PROGRAM OP160_Initialization_Seq
VAR
	op160_master_reset :BOOL;
	op160_robot_homed  :BOOL;
	op160_ROboProgResetDly   :ton;
END_VAR

IF CR160_MoverREM_Cyl.Position1 AND OP160_SO_Rbt_In_Home AND op160_robot_homed THEN
   OP160_Temp_Home_OK:=TRUE;
ELSE
	OP160_Temp_Home_OK:=FALSE;
END_IF

IF OP160_ErrorActive THEN 
	op160_robot_homed    :=FALSE;
END_IF

CASE OP160_Homing_Seq OF
	
	0: IF (OP160_Auto AND NOT OP160_HomeRunning AND  NOT OP160_ErrorActive AND  NOT 
			OP160_AutoRunning AND NOT OP160_StepRunning	 AND NOT OP160_Temp_Home_OK) THEN
		    OP160_HomeRunning:=TRUE;
		    OP160_Homing_Seq:=10;	
	   END_IF
	   
	10:IF (OP160_HomeRunning AND OP160_HMI_Homing)THEN
		OP160_Homing_Seq:=12;		
		END_IF 
        
	
   12:  OP160_Robo_ProgramReset:=TRUE;
   
		IF NOT OP160_SO_Program_Execute	AND op160_ROboProgResetDly.Q THEN
		OP160_Robo_ProgramReset:=FALSE;			
		OP160_Homing_Seq:=14;	
		END_IF
	
		
	
	14: IF OP160_HomeRunning AND NOT op160_master_reset THEN
		   OP160_Robo_Out6001   :=1;
	       OP160_SI_Homing_Start:=TRUE;
	       OP160_Homing_Seq:=15;
	    
		ELSIF  OP160_HomeRunning AND  op160_master_reset THEN
		       OP160_Robo_Out6001   :=3;
	           OP160_SI_Homing_Start:=TRUE;
	           OP160_Homing_Seq     :=15;
		END_IF
		
		
      (*  OP160_Robo_Out6001:=3;
        
		IF OP160_SO_Rbt_In_Home THEN
		OP160_SI_Homing_Start:=FALSE;
		
		OP160_Robo_ProgramReset:=TRUE;	
		END_IF
		IF NOT OP160_SO_Program_Execute	AND OP160_Robo_ProgramReset=TRUE THEN
		OP160_Robo_ProgramReset:=FALSE;
		OP160_Homing_Seq:=20;		
		END_IF *)
			
	15: IF OP160_HomeRunning AND OP160_SO_Rbt_In_Home THEN
		   OP160_SI_Homing_Start:=FALSE;
		   op160_robot_homed    :=TRUE;
		   OP160_Homing_Seq:=20;
	    END_IF
 
	
	20:IF (OP160_HomeRunning AND OP160_HMI_Homing)THEN 
        IF ( CR160_MoverREM_Cyl.Position1 ) THEN
			OP160_Homing_Seq:=30;
		ELSE
			CR160_MoverREM_Cyl.HomingCmd1:= TRUE;
				
		END_IF
		END_IF
	
		
	30:	OP160_Homing_Seq:=0;
		OP160_HomeRunning:=FALSE;
	
END_CASE

IF NOT OP160_HomeRunning THEN
	CR160_MoverREM_Cyl.HomingCmd1:= FALSE;
END_IF

op160_ROboProgResetDly(IN:= OP160_Robo_ProgramReset, PT:= T#200MS, Q=> , ET=> );

END_PROGRAM

(* stored: Version 1.1.0.1, ProductVersion 3.1.4024.11
   POU OP160_Initialization_Seq: Id {dbee5b30-95ec-4991-8753-6971fcbddff0}, SpecialFunc None *)
